PROGRAM EM05_PlacingArea_4
VAR
//----Motor-----
	// Box Placing Roller Conveyor 4	
	FB_BoxPlacingRollerConv_4					: MotorManagement;
	stBoxPlacingRollerConv_4					: stMotor;
	BoxPlacingRollerConv_4_ErrorID				: UINT;
	BoxPlacingRollerConv_4_Error				: BOOL;
	bFL_BoxPlacingRollerConv_4_Forward			: BOOL;
	bFL_BoxPlacingRollerConv_4_Reverse			: BOOL;
	// Empty And Load Transfer Roller Conveyor 	
	FB_EmptyAndLoadTransferRollerConv			: MotorManagement;
	stEmptyAndLoadTransferRollerConv			: stMotor;
	EmptyAndLoadTransferRollerConv_ErrorID		: UINT;
	EmptyAndLoadTransferRollerConv_Error		: BOOL;
	bFL_EmptyAndLoadTransferRollerConv_Forward	: BOOL;
	bFL_EmptyAndLoadTransferRollerConv_Reverse	: BOOL;
	// Empty And Load Turning Conveyor 1	
	FB_EmptyAndLoadTurningConv_1				: MotorManagement;
	stEmptyAndLoadTurningConv_1					: stMotor;
	EmptyAndLoadTurningConv_1_ErrorID			: UINT;
	EmptyAndLoadTurningConv_1_Error				: BOOL;
	bFL_EmptyAndLoadTurningConv_1_Forward		: BOOL;
	bFL_EmptyAndLoadTurningConv_1_Reverse		: BOOL;
	// Empty And Load Turning Conveyor 2	
	FB_EmptyAndLoadTurningConv_2				: MotorManagement;
	stEmptyAndLoadTurningConv_2					: stMotor;
	EmptyAndLoadTurningConv_2_ErrorID			: UINT;
	EmptyAndLoadTurningConv_2_Error				: BOOL;
	bFL_EmptyAndLoadTurningConv_2_Forward		: BOOL;
	bFL_EmptyAndLoadTurningConv_2_Reverse		: BOOL;
END_VAR

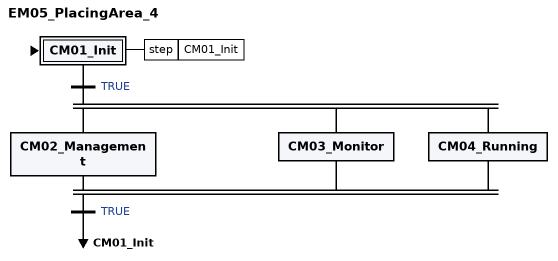
INITIAL_STEP CM01_Init:
    CM01_Init(N);  // step action
END_STEP
TRANSITION FROM CM01_Init TO (CM02_Management, CM03_Monitor, CM04_Running)
    := TRUE;
END_TRANSITION
STEP CM02_Management:
END_STEP
STEP CM03_Monitor:
END_STEP
STEP CM04_Running:
END_STEP
TRANSITION FROM (CM02_Management, CM03_Monitor, CM04_Running) TO CM01_Init
    := TRUE;
END_TRANSITION

ACTION CM01_Init:

END_ACTION

ACTION CM02_Management:
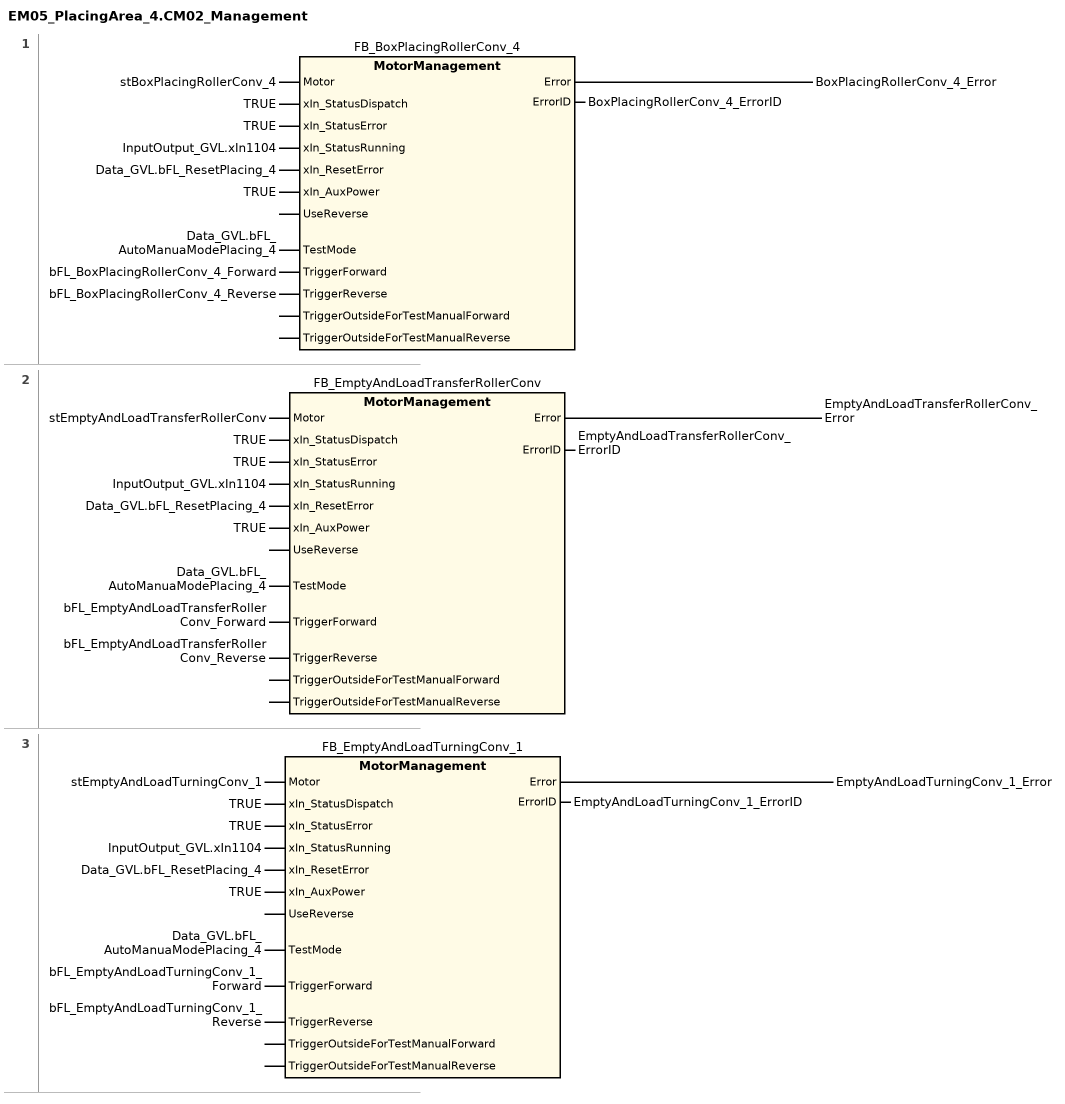
// NETWORK 1
FB_BoxPlacingRollerConv_4(
    Motor := stBoxPlacingRollerConv_4,
    xIn_StatusDispatch := TRUE,
    xIn_StatusError := TRUE,
    xIn_StatusRunning := InputOutput_GVL.xIn1104,
    xIn_ResetError := Data_GVL.bFL_ResetPlacing_4,
    xIn_AuxPower := TRUE,
    TestMode := Data_GVL.bFL_AutoManuaModePlacing_4,
    TriggerForward := bFL_BoxPlacingRollerConv_4_Forward,
    TriggerReverse := bFL_BoxPlacingRollerConv_4_Reverse,
    ErrorID => BoxPlacingRollerConv_4_ErrorID); // MotorManagement
BoxPlacingRollerConv_4_Error := FB_BoxPlacingRollerConv_4.Error;

// NETWORK 2
FB_EmptyAndLoadTransferRollerConv(
    Motor := stEmptyAndLoadTransferRollerConv,
    xIn_StatusDispatch := TRUE,
    xIn_StatusError := TRUE,
    xIn_StatusRunning := InputOutput_GVL.xIn1104,
    xIn_ResetError := Data_GVL.bFL_ResetPlacing_4,
    xIn_AuxPower := TRUE,
    TestMode := Data_GVL.bFL_AutoManuaModePlacing_4,
    TriggerForward := bFL_EmptyAndLoadTransferRollerConv_Forward,
    TriggerReverse := bFL_EmptyAndLoadTransferRollerConv_Reverse,
    ErrorID => EmptyAndLoadTransferRollerConv_ErrorID); // MotorManagement
EmptyAndLoadTransferRollerConv_Error := FB_EmptyAndLoadTransferRollerConv.Error;

// NETWORK 3
FB_EmptyAndLoadTurningConv_1(
    Motor := stEmptyAndLoadTurningConv_1,
    xIn_StatusDispatch := TRUE,
    xIn_StatusError := TRUE,
    xIn_StatusRunning := InputOutput_GVL.xIn1104,
    xIn_ResetError := Data_GVL.bFL_ResetPlacing_4,
    xIn_AuxPower := TRUE,
    TestMode := Data_GVL.bFL_AutoManuaModePlacing_4,
    TriggerForward := bFL_EmptyAndLoadTurningConv_1_Forward,
    TriggerReverse := bFL_EmptyAndLoadTurningConv_1_Reverse,
    ErrorID => EmptyAndLoadTurningConv_1_ErrorID); // MotorManagement
EmptyAndLoadTurningConv_1_Error := FB_EmptyAndLoadTurningConv_1.Error;

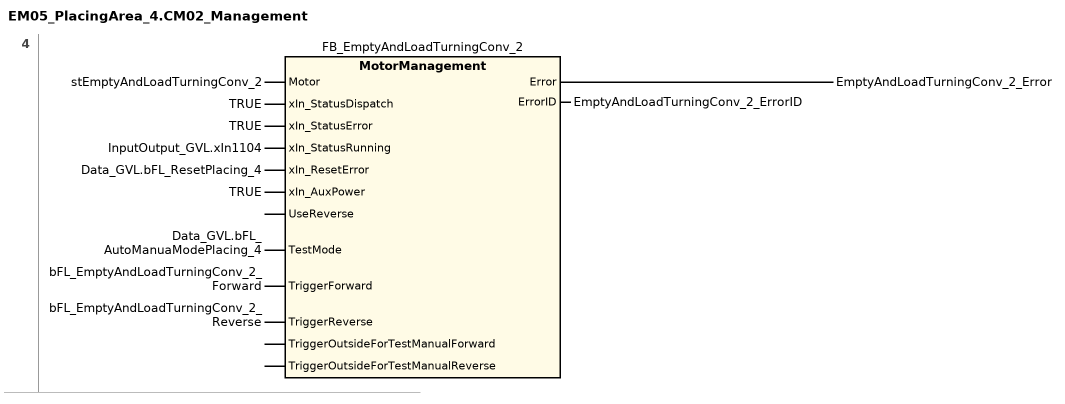
// NETWORK 4
FB_EmptyAndLoadTurningConv_2(
    Motor := stEmptyAndLoadTurningConv_2,
    xIn_StatusDispatch := TRUE,
    xIn_StatusError := TRUE,
    xIn_StatusRunning := InputOutput_GVL.xIn1104,
    xIn_ResetError := Data_GVL.bFL_ResetPlacing_4,
    xIn_AuxPower := TRUE,
    TestMode := Data_GVL.bFL_AutoManuaModePlacing_4,
    TriggerForward := bFL_EmptyAndLoadTurningConv_2_Forward,
    TriggerReverse := bFL_EmptyAndLoadTurningConv_2_Reverse,
    ErrorID => EmptyAndLoadTurningConv_2_ErrorID); // MotorManagement
EmptyAndLoadTurningConv_2_Error := FB_EmptyAndLoadTurningConv_2.Error;
END_ACTION

ACTION CM03_Monitor:
// NETWORK 1
END_ACTION

ACTION CM04_Running:
// NETWORK 1
END_ACTION

END_PROGRAM

(* stored: Version 1.1.0.1, ProductVersion 3.1.4024.9
   POU EM05_PlacingArea_4: Id {0bb07f72-b5fb-4837-9881-8ca1fe874c00}, SpecialFunc None
   Action CM01_Init: Id {042b9ee1-f4a0-4633-a8a1-88a8bebccea5}
   Action CM02_Management: Id {37bc2a98-748c-4983-b53d-0141c7b0a713}
   Action CM03_Monitor: Id {cbdc493e-f475-4cae-823b-1116a94210a9}
   Action CM04_Running: Id {31eb77bc-8b8b-4bea-b96c-3c5dfd3a817c} *)
